(* Logix 5000 project; controller PBS_Perfusion vendor 1 type 14 code 217 rev 32.14; software revision 32.03; part 16 of 27 *)
(* tags used below, declared in another part *)
   Inp_IOFault : BOOL;   // Input Communication Status 0=OK, 1=fail
   Inp_Sim : BOOL;   // 1=Simulate working device; 0=Turn ON/OFF actual device
   Inp_OvrdCmd : DINT;   // Ovrd Device Command 0=None, 1=Off, 2=On, 3=Pulse Off, 4=Pulse On, 5=Pulse Cont
   Cfg_HasOnFdbk : BOOL;   // 1=Device provides an ON feedback signal
   Cfg_HasOffFdbk : BOOL;   // 1=Device provides an OFF feedback signal
   PSet_Owner : DINT;   // Program Owner Request ID (non-zero) or Release (zero)
   PCmd_On : BOOL;   // Program Command to turn device ON
   PCmd_Off : BOOL;   // Program Command to turn device OFF
   PCmd_OnPulse : BOOL;   // Program Command to pulse device (which is OFF) ON once
   PCmd_OffPulse : BOOL;   // Program Command to pulse device (which is ON) OFF once
   PCmd_ContPulse : BOOL;   // Program Command to pulse device continuously (blink)
   XCmd_On : BOOL;   // External Command to turn device ON
   XCmd_Off : BOOL;   // External Command to turn device OFF
   XCmd_OnPulse : BOOL;   // External Command to pulse device (which is OFF) ON once
   XCmd_OffPulse : BOOL;   // External Command to pulse device (which is ON) OFF once
   XCmd_ContPulse : BOOL;   // External Command to pulse device continuously (blink)
   XCmd_Reset : BOOL;   // Ext Cmd to clear shed latches and cleared alarms
   Out_Horn : BOOL;   // 1=Sound audible prior to commanded energize/ state change
   SrcQ_IO : DINT;   // Source and Quality of primary I/O (enumeration)
   SrcQ : DINT;   // Source and Quality of primary Val/Sts (enumeration)
   Val_Cmd : DINT;   // Device Command: 0=None, 1=Off, 2=On, 3=Pulse Off, 4=Pulse On, 5=Pulse Cont
   Val_Sts : DINT;   // Device Status 0=off 1=on 2=pulse off 3=pulse on 4=pulse cont. 5=turning off 6=turning on
   Val_Fault : DINT;   // Device Fault Status 0=none, 16=Feedback Fault, 32=I/O Fault, 34=Config Error
   Val_State : DINT;   // Internal Logic State (for animating STD on faceplate), see manual
   Val_NotifyAll : DINT;   // Highest Alarm prio and ack status this object + attached (enum)
   Val_UnackAlmC : DINT;   // Count of Unacknowledged Alarms
   Val_Owner : DINT;   // Current Object Owner ID (0=not owned)
   Sts_Out : BOOL;   // 1=Output is ON (energized), 0=Output is OFF (de-energized)
   Sts_Horn : BOOL;   // 1=Horn Active
   Nrdy_CfgErr : BOOL;   // 1=Device Not Ready: Configuration Error
   Nrdy_Fail : BOOL;   // 1=Device Not Ready: Device Failure (Shed Requires Reset)
   Nrdy_IOFault : BOOL;   // 1=Device Not Ready: I/O Fault (Shed Requires Reset)
   Nrdy_PrioOff : BOOL;   // 1=Device Not Ready: Oper/Ext Priority Off Comand Requires Reset
   Sts_AlmInh : BOOL;   // 1=One or more Alarms Shelved, Disabled or Suppressed
   Err_Alarm : BOOL;   // 1=Error in Config: Alarm Min On Time, Shelf Time, Severity
   Sts_OoS : ALIAS FOR CmdSrc.Sts_OoS;
   Sts_RdyAck : BOOL;   // 1=An alarm is ready to be acknowledged
   Sts_OnFail : ALIAS FOR OnFail.Inp;   // 1=Device Failed to Turn ON
   Sts_OffFail : ALIAS FOR OffFail.Inp;   // 1=Device Failed to Turn OFF
   Sts_IOFault : ALIAS FOR IOFault.Inp;   // I/O Comm Fault Status (0=OK, 1=Bad)
   P_DOut : BOOL;   // Unique Parameter Name for auto - discovery
   Wrk_Notify : DINT;   // Buffer for building Val_Notify
   CmdSrc : P_CmdSrc;   // Control / Command Source Selection
   IOFault : P_Alarm;   // I/O Fault Alarm
   IntlkTrip : P_Alarm;   // Interlock Trip Alarm
   OffFail : P_Alarm;   // Device Failed to Turn OFF Alarm
   OnFail : P_Alarm;   // Device Failed to Turn ON Alarm
   Wrk_Cmd : DINT;   // Device Command: 0= None, bit .0=Off, bit .1=On, bit .2=Pulse Off, bit .3=Pulse On, bit .4=Pulse Cont.
   Wrk_Fault : DINT;   // Buffer for building Val_Fault
   Wrk_SrcQ : DINT;   // Register for building Source / Quality enumeration
   Wrk_UnackAlmC : DINT;   // Buffer for building Val_UnackAlmC
   Val_Notify : DINT;   // Current Alarm Level and Acknowledgement (enumeration)
   OCmd_ResetAckAll : BOOL;   // Operator Command to Reset all Alarms and latched Shed conditions
   OCmd_ContPulse : BOOL;   // Operator Command to pulse device continuously (blink)
   OCmd_OffPulse : BOOL;   // Operator Command to pulse device (which is ON) OFF once
   OCmd_OnPulse : BOOL;   // Operator Command to pulse device (which is OFF) ON once
   OCmd_Off : BOOL;   // Operator Command to turn device OFF
   OCmd_On : BOOL;   // Operator Command to turn device ON
   MCmd_Check : BOOL;   // Maintenance Command to Check (not bypass) all Interlocks and Permissives
   MCmd_Bypass : BOOL;   // Maintenance Command to Bypass all Bypassable Interlocks and Permissives
   ORdy_ResetAckAll : BOOL;   // 1=Ready for OCmd_ResetAckAll (enables HMI button)
   ORdy_ContPulse : BOOL;   // 1=Ready for OCmd_ContPulse (enables HMI button)
   ORdy_OffPulse : BOOL;   // 1=Ready for OCmd_OffPulse (enables HMI button)
   ORdy_OnPulse : BOOL;   // 1=Ready for OCmd_OnPulse (enables HMI button)
   ORdy_Off : BOOL;   // 1=Ready for OCmd_Off (enables HMI button)
   ORdy_On : BOOL;   // 1=Ready for OCmd_On (enables HMI button)
   MRdy_Check : BOOL;   // 1=Ready for MCmd_Check (enables HMI button)
   MRdy_Bypass : BOOL;   // 1=Ready for MCmd_Bypass (enables HMI button)
   Wrk_State : DINT;   // Internal value of state machine current state
   Wrk_StartHorn : BOOL;   // 1=Sound audible prior to commanded energize/ state change
   ONS : DINT[3];
   REAL : DINT;
(* P_DOut, continued *)

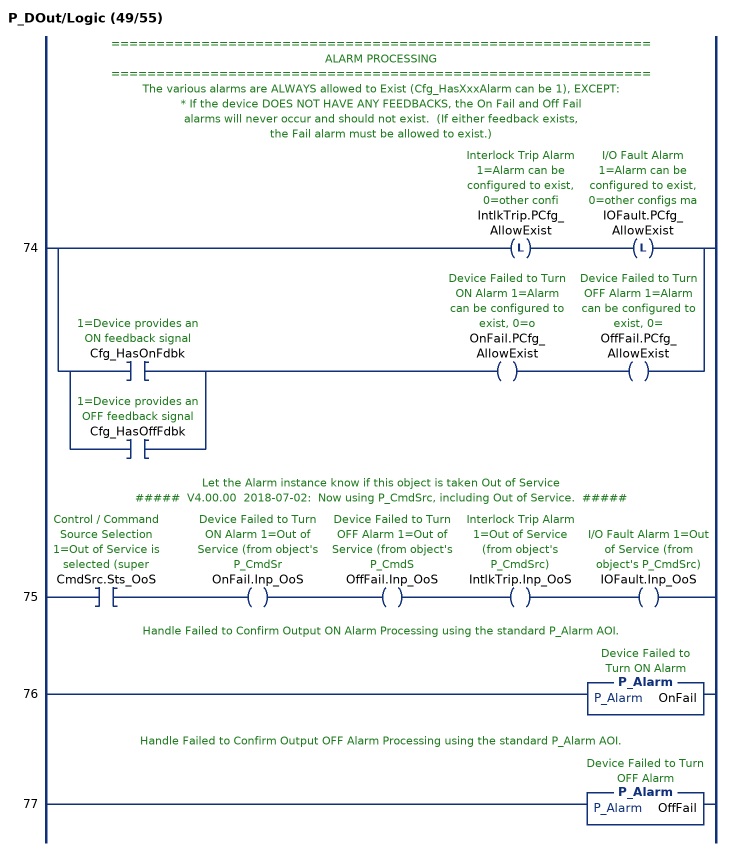
   // ============================================================
   // ALARM PROCESSING
   // ============================================================
   // The various alarms are ALWAYS allowed to Exist (Cfg_HasXxxAlarm can be 1), EXCEPT:
   // * If the device DOES NOT HAVE ANY FEEDBACKS, the On Fail and Off Fail
   // alarms will never occur and should not exist.  (If either feedback exists,
   // the Fail alarm must be allowed to exist.)
   74: [OTL(IntlkTrip.PCfg_AllowExist) OTL(IOFault.PCfg_AllowExist) ,[XIC(Cfg_HasOnFdbk) ,XIC(Cfg_HasOffFdbk) ] OTE(OnFail.PCfg_AllowExist) OTE(OffFail.PCfg_AllowExist) ];
   // Let the Alarm instance know if this object is taken Out of Service
   // #####  V4.00.00  2018-07-02:  Now using P_CmdSrc, including Out of Service.  #####
   75: XIC(CmdSrc.Sts_OoS)OTE(OnFail.Inp_OoS)OTE(OffFail.Inp_OoS)OTE(IntlkTrip.Inp_OoS)OTE(IOFault.Inp_OoS);
   // Handle Failed to Confirm Output ON Alarm Processing using the standard P_Alarm AOI.
   76: P_Alarm(OnFail);
   // Handle Failed to Confirm Output OFF Alarm Processing using the standard P_Alarm AOI.
   77: P_Alarm(OffFail);
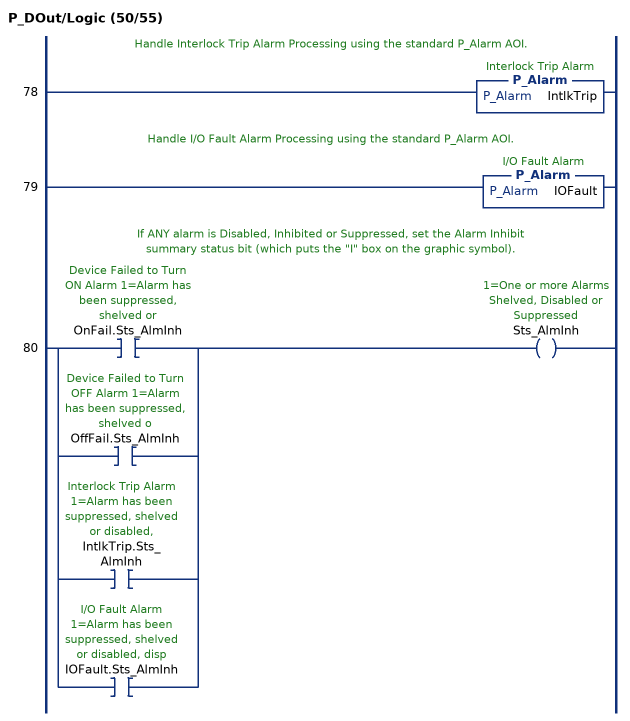
   // Handle Interlock Trip Alarm Processing using the standard P_Alarm AOI.
   78: P_Alarm(IntlkTrip);
   // Handle I/O Fault Alarm Processing using the standard P_Alarm AOI.
   79: P_Alarm(IOFault);
   // If ANY alarm is Disabled, Inhibited or Suppressed, set the Alarm Inhibit
   // summary status bit (which puts the "I" box on the graphic symbol).
   80: [XIC(OnFail.Sts_AlmInh) ,XIC(OffFail.Sts_AlmInh) ,XIC(IntlkTrip.Sts_AlmInh) ,XIC(IOFault.Sts_AlmInh) ]OTE(Sts_AlmInh);
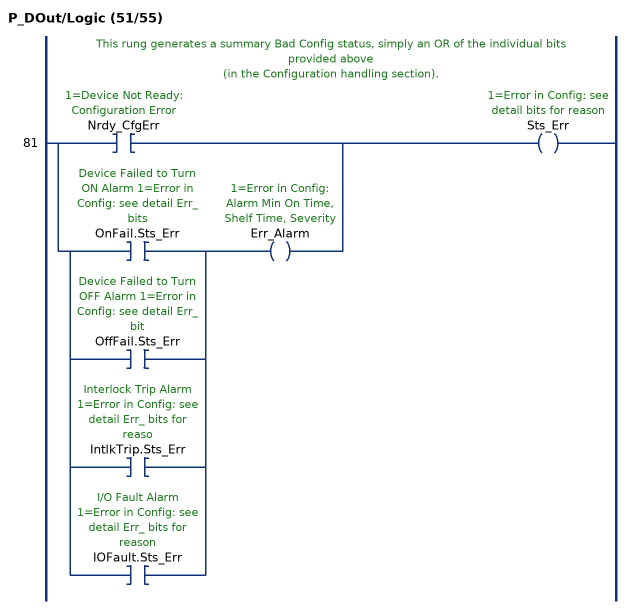
   // This rung generates a summary Bad Config status, simply an OR of the individual bits provided above
   // (in the Configuration handling section).
   81: [XIC(Nrdy_CfgErr) ,[XIC(OnFail.Sts_Err) ,XIC(OffFail.Sts_Err) ,XIC(IntlkTrip.Sts_Err) ,XIC(IOFault.Sts_Err) ] OTE(Err_Alarm) ]OTE(Sts_Err);
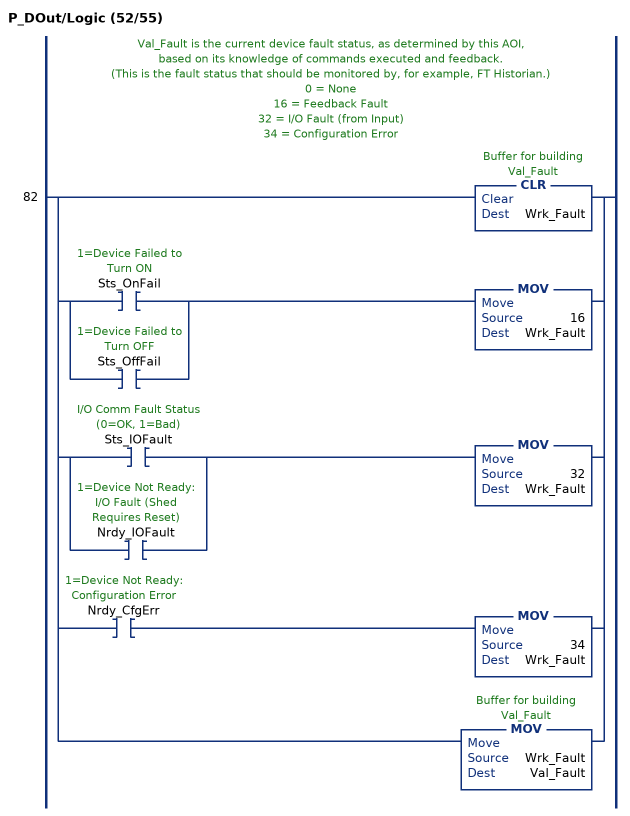
   // Val_Fault is the current device fault status, as determined by this AOI,
   // based on its knowledge of commands executed and feedback.
   // (This is the fault status that should be monitored by, for example, FT Historian.)
   // 0 = None
   // 16 = Feedback Fault
   // 32 = I/O Fault (from Input)
   // 34 = Configuration Error
   82: [CLR(Wrk_Fault) ,[XIC(Sts_OnFail) ,XIC(Sts_OffFail) ] MOV(16,Wrk_Fault) ,[XIC(Sts_IOFault) ,XIC(Nrdy_IOFault) ] MOV(32,Wrk_Fault) ,XIC(Nrdy_CfgErr) MOV(34,Wrk_Fault) ,MOV(Wrk_Fault,Val_Fault) ];
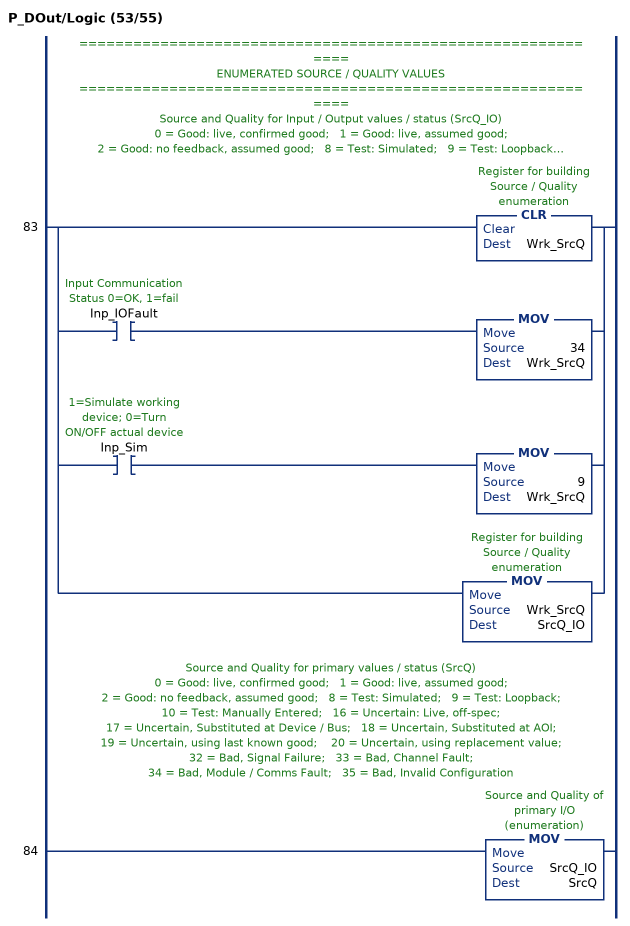
   // ============================================================
   // ENUMERATED SOURCE / QUALITY VALUES
   // ============================================================
   // Source and Quality for Input / Output values / status (SrcQ_IO)
   // 0 = Good: live, confirmed good;   1 = Good: live, assumed good;
   // 2 = Good: no feedback, assumed good;   8 = Test: Simulated;   9 = Test: Loopback;
   // 10 = Test: Manually Entered;   16 = Uncertain: Live, off-spec;
   // 17 = Uncertain, Substituted at Device / Bus;   18 = Uncertain, Substituted at AOI;
   // 19 = Uncertain, using last known good;    20 = Uncertain, using replacement value;
   // 32 = Bad, Signal Failure;   33 = Bad, Channel Fault;
   // 34 = Bad, Module / Comms Fault;   35 = Bad, Invalid Configuration
   83: [CLR(Wrk_SrcQ) ,XIC(Inp_IOFault) MOV(34,Wrk_SrcQ) ,XIC(Inp_Sim) MOV(9,Wrk_SrcQ) ,MOV(Wrk_SrcQ,SrcQ_IO) ];
   // Source and Quality for primary values / status (SrcQ)
   // 0 = Good: live, confirmed good;   1 = Good: live, assumed good;
   // 2 = Good: no feedback, assumed good;   8 = Test: Simulated;   9 = Test: Loopback;
   // 10 = Test: Manually Entered;   16 = Uncertain: Live, off-spec;
   // 17 = Uncertain, Substituted at Device / Bus;   18 = Uncertain, Substituted at AOI;
   // 19 = Uncertain, using last known good;    20 = Uncertain, using replacement value;
   // 32 = Bad, Signal Failure;   33 = Bad, Channel Fault;
   // 34 = Bad, Module / Comms Fault;   35 = Bad, Invalid Configuration
   84: MOV(SrcQ_IO,SrcQ);
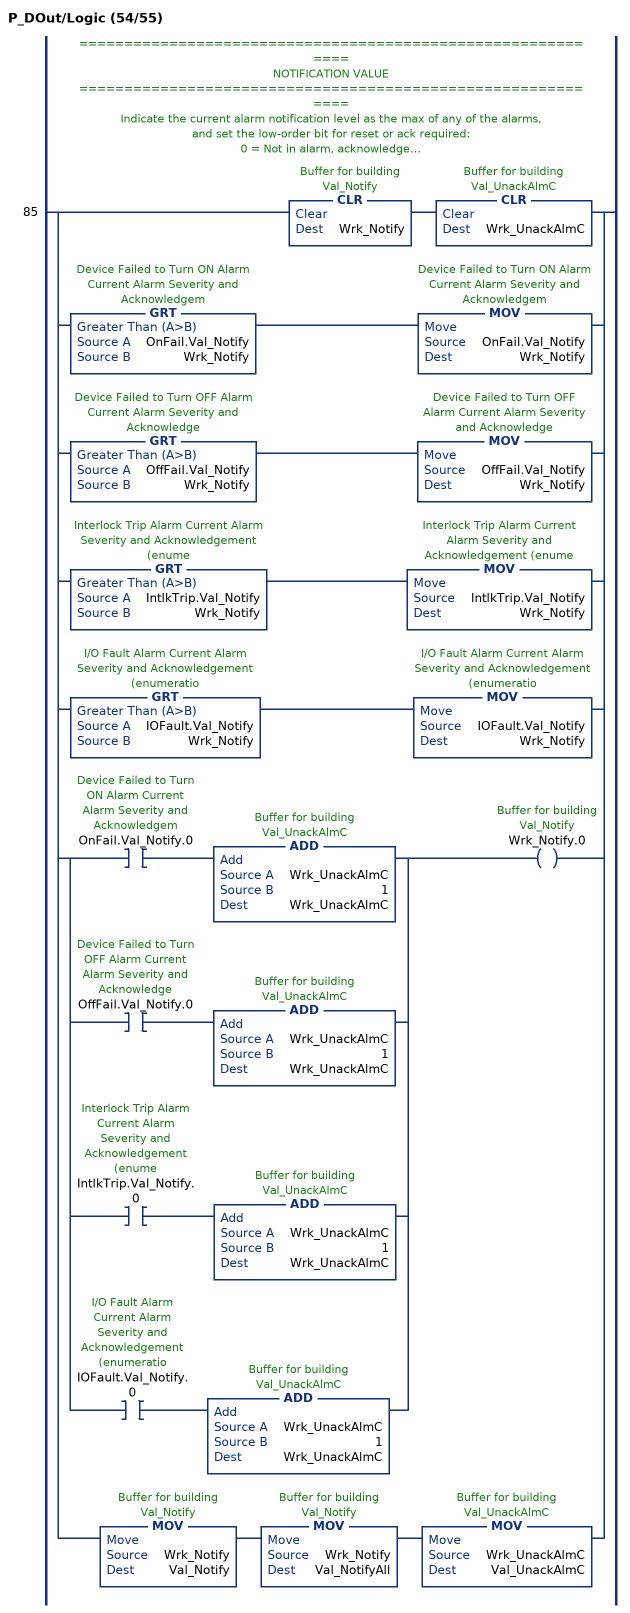
   // ============================================================
   // NOTIFICATION VALUE
   // ============================================================
   // Indicate the current alarm notification level as the max of any of the alarms,
   // and set the low-order bit for reset or ack required:
   // 0 = Not in alarm, acknowledged
   // 1 = Not in alarm, unacknowledged or reset required
   // 2 = Low severity alarm, acknowledged
   // 3 = Low severity alarm, unacknowledged
   // 4 = Medium severity alarm, acknowledged
   // 5 = Medium severity alarm, unacknowledged
   // 6 = High severity alarm, acknowledged
   // 7 = High severity alarm, unacknowledged
   // 8 = Urgent severity alarm, acknowledged
   // 9 = Urgent severity alarm, unacknowledged
   // #####  V4.00.00  2018-07-02:  Added Val_NotifyAll and Val_UnackAlmC to roll up alarm  #####
   // #####  priority / ack status and unack. alarm count.  #####
   85: [CLR(Wrk_Notify) CLR(Wrk_UnackAlmC) ,GRT(OnFail.Val_Notify,Wrk_Notify) MOV(OnFail.Val_Notify,Wrk_Notify) ,GRT(OffFail.Val_Notify,Wrk_Notify) MOV(OffFail.Val_Notify,Wrk_Notify) ,GRT(IntlkTrip.Val_Notify,Wrk_Notify) MOV(IntlkTrip.Val_Notify,Wrk_Notify) ,GRT(IOFault.Val_Notify,Wrk_Notify) MOV(IOFault.Val_Notify,Wrk_Notify) ,[XIC(OnFail.Val_Notify.0) ADD(Wrk_UnackAlmC,1,Wrk_UnackAlmC) ,XIC(OffFail.Val_Notify.0) ADD(Wrk_UnackAlmC,1,Wrk_UnackAlmC) ,XIC(IntlkTrip.Val_Notify.0) ADD(Wrk_UnackAlmC,1,Wrk_UnackAlmC) ,XIC(IOFault.Val_Notify.0) ADD(Wrk_UnackAlmC,1,Wrk_UnackAlmC) ] OTE(Wrk_Notify.0) ,MOV(Wrk_Notify,Val_Notify) MOV(Wrk_Notify,Val_NotifyAll) MOV(Wrk_UnackAlmC,Val_UnackAlmC) ];
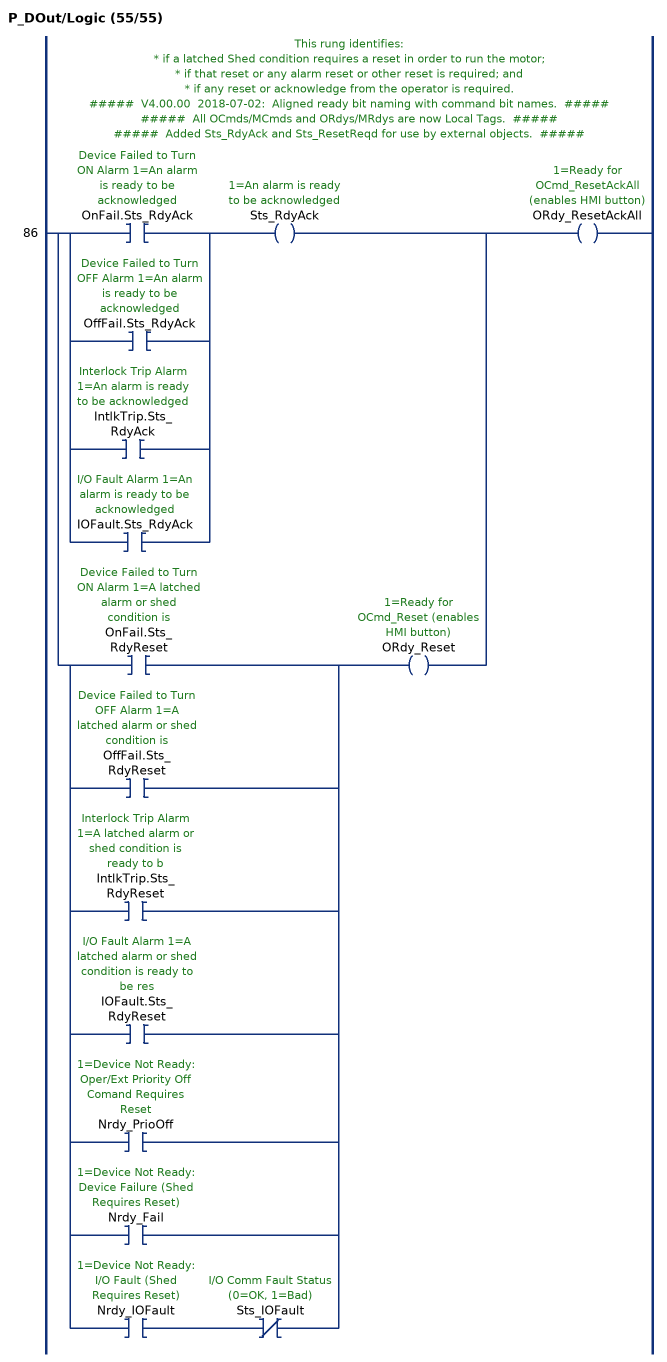
   // This rung identifies:
   // * if a latched Shed condition requires a reset in order to run the motor;
   // * if that reset or any alarm reset or other reset is required; and
   // * if any reset or acknowledge from the operator is required.
   // #####  V4.00.00  2018-07-02:  Aligned ready bit naming with command bit names.  #####
   // #####  All OCmds/MCmds and ORdys/MRdys are now Local Tags.  #####
   // #####  Added Sts_RdyAck and Sts_ResetReqd for use by external objects.  #####
   86: [[XIC(OnFail.Sts_RdyAck) ,XIC(OffFail.Sts_RdyAck) ,XIC(IntlkTrip.Sts_RdyAck) ,XIC(IOFault.Sts_RdyAck) ] OTE(Sts_RdyAck) ,[XIC(OnFail.Sts_RdyReset) ,XIC(OffFail.Sts_RdyReset) ,XIC(IntlkTrip.Sts_RdyReset) ,XIC(IOFault.Sts_RdyReset) ,XIC(Nrdy_PrioOff) ,XIC(Nrdy_Fail) ,XIC(Nrdy_IOFault) XIO(Sts_IOFault) ] OTE(ORdy_Reset) ]OTE(ORdy_ResetAckAll);
END_ROUTINE

ROUTINE Prescan   (* ladder *)
// Clear Ownershp, clear "lurking" Commands, de-energize output
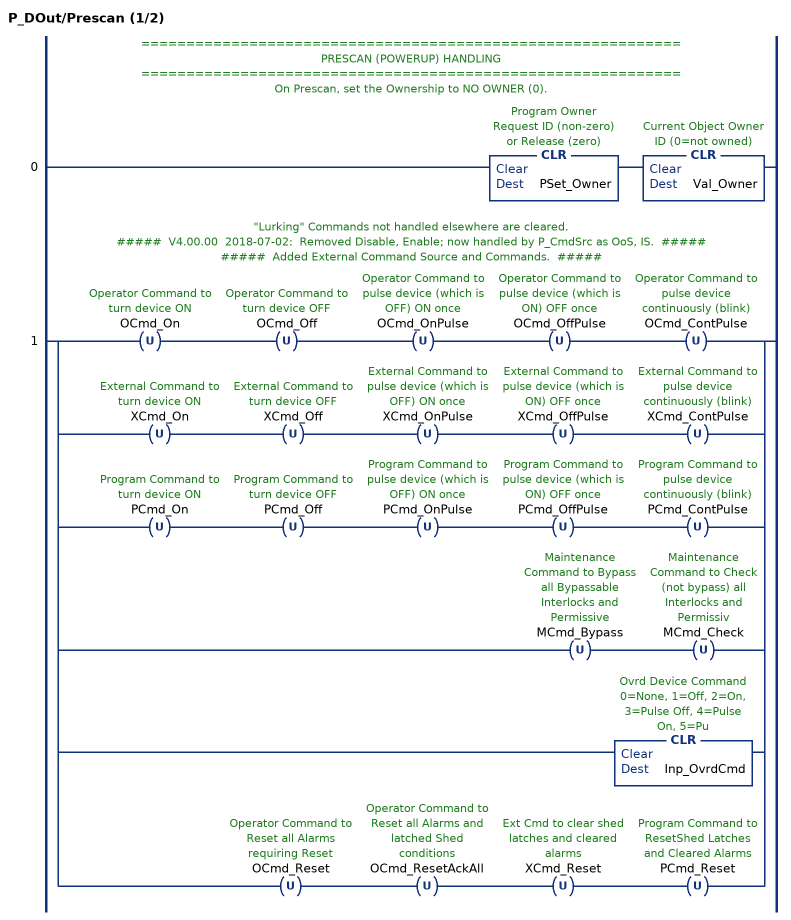
   // ============================================================
   // PRESCAN (POWERUP) HANDLING
   // ============================================================
   // On Prescan, set the Ownership to NO OWNER (0).
   0: CLR(PSet_Owner)CLR(Val_Owner);
   // "Lurking" Commands not handled elsewhere are cleared.
   // #####  V4.00.00  2018-07-02:  Removed Disable, Enable; now handled by P_CmdSrc as OoS, IS.  #####
   // #####  Added External Command Source and Commands.  #####
   1: [OTU(OCmd_On) OTU(OCmd_Off) OTU(OCmd_OnPulse) OTU(OCmd_OffPulse) OTU(OCmd_ContPulse) ,OTU(XCmd_On) OTU(XCmd_Off) OTU(XCmd_OnPulse) OTU(XCmd_OffPulse) OTU(XCmd_ContPulse) ,OTU(PCmd_On) OTU(PCmd_Off) OTU(PCmd_OnPulse) OTU(PCmd_OffPulse) OTU(PCmd_ContPulse) ,OTU(MCmd_Bypass) OTU(MCmd_Check) ,CLR(Inp_OvrdCmd) ,OTU(OCmd_Reset) OTU(OCmd_ResetAckAll) OTU(XCmd_Reset) OTU(PCmd_Reset) ];
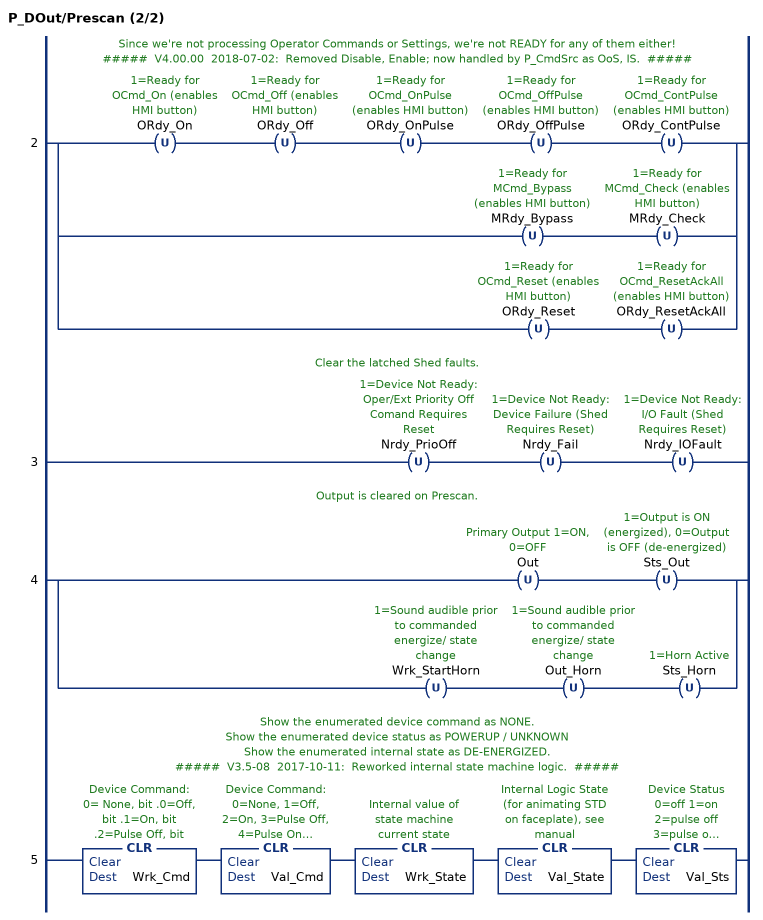
   // Since we're not processing Operator Commands or Settings, we're not READY for any of them either!
   // #####  V4.00.00  2018-07-02:  Removed Disable, Enable; now handled by P_CmdSrc as OoS, IS.  #####
   2: [OTU(ORdy_On) OTU(ORdy_Off) OTU(ORdy_OnPulse) OTU(ORdy_OffPulse) OTU(ORdy_ContPulse) ,OTU(MRdy_Bypass) OTU(MRdy_Check) ,OTU(ORdy_Reset) OTU(ORdy_ResetAckAll) ];
   // Clear the latched Shed faults.
   3: OTU(Nrdy_PrioOff)OTU(Nrdy_Fail)OTU(Nrdy_IOFault);
   // Output is cleared on Prescan.
   4: [OTU(Out) OTU(Sts_Out) ,OTU(Wrk_StartHorn) OTU(Out_Horn) OTU(Sts_Horn) ];
   // Show the enumerated device command as NONE.
   // Show the enumerated device status as POWERUP / UNKNOWN
   // Show the enumerated internal state as DE-ENERGIZED.
   // #####  V3.5-08  2017-10-11:  Reworked internal state machine logic.  #####
   5: CLR(Wrk_Cmd)CLR(Val_Cmd)CLR(Wrk_State)CLR(Val_State)CLR(Val_Sts);
END_ROUTINE
END_ADD_ON_INSTRUCTION

ADD_ON_INSTRUCTION P_Gate   (* revision 4.10 .00 Release, vendor Rockwell Automation, ExecutePrescan, ExecuteEnableInFalse *)
// Condition Gate/Delay
// Revision note:
// See Instruction Help for a summary of changes, and see 4.10 Release Notes for details.
// Help:
// Copyright © Rockwell Automation, Inc.  All Rights Reserved.
// This Instruction provides a "gate" for a discrete Input signal and
// provides on-delay and off-delay timing for the gated signal.
// When the Gate input is true, the instruction Input is passed through
// to the Output, with on-delay and off-delay timing applied.
// When the Gate input is false, the Output is kept off
// (note: off-delay still applies!)
// This instruction is usually used between a comparison
// (analog threshold with deadband or discrete logic)
// and a P_Alarm instance, but may be used as a
// gated on-delay/off-delay timer generally.
// When EnableIn  is FALSE (e.g., on a false LD rung), the Input "Inp"
// is inverted.  Note that the Gate input (Inp_Gate) is NOT inverted!!!
// SUMMARY OF CHANGES FROM PREVIOUS VERSION (4.00.00)
// See 4.10 Release Notes for details.
// * Unmodified, up-rev only for Library 4.10.00
// SUMMARY OF CHANGES FROM PREVIOUS VERSION (3.5-01)
// See 4.00 Release Notes for details.
// * Changed Inf_ items to HMI_ (e.g., HMI_Lib, HMI_Type).
// * Changed delay time configuration items to REAL seconds
VAR_INPUT
   Inp : BOOL; {visible}   // Input Condition: e.g., result of comparison
   Inp_Gate : BOOL := 1; {visible}   // Gate Input: 1=enable On Delay / Off Delay after Gate Delay, 0=disable
   Cfg_GateDly : REAL;   // Gate Delay (s): time after Gate Input true to enable On/Off Delay
   Cfg_OnDly : REAL;   // On Delay (s): If Gate Delay done, time Inp must be true to set Out true
   Cfg_OffDly : REAL;   // Off Delay (s): Time after Inp or Gate goes to 0 for Out to go to 0
END_VAR
VAR_OUTPUT
   Out : BOOL; {access Read Only, visible}   // Output after On Delay, Off Delay, enabled by Gate
   Sts_Gate : BOOL; {access Read Only, visible}   // 1=Gate Delay done, Output is enabled
   Sts_Err : BOOL; {access Read Only, visible}   // 1=Error in Config (see detail Err_ bits for reason), display icon
   Err_Timer : BOOL; {access Read Only}   // 1=Error in Config: On Delay, Off Delay, Gate Delay Time Invalid (use 0 to 2147483 s)
   P_Gate : BOOL;   // Unique Parameter Name for auto - discovery
END_VAR
VAR
   Wrk_OffDlyT : TIMER; {access Read Only}   // Off Delay Timer
   Wrk_OnDlyT : TIMER; {access Read Only}   // On Delay Timer
   Wrk_GateT : TIMER; {access Read Only}   // Gate Delay Timer
   Cfg_InpCond : STRING_20 := 'Input Condition';   // Displayed text of P_Gate's Input (Inp) Condition
   HMI_Lib : STRING_12 := 'RA-BAS'; {access Read Only}   // Display Library for Faceplate call-up
   HMI_Type : STRING_16 := 'P_Gate'; {access Read Only}   // Must contain AOI name, used for HMI and Information S/W
   Cfg_GateCond : STRING_20 := 'Gating Condition';   // Displayed text of P_Gate's Gating (Inp_Gate) Condition
   HMI_Tab : SINT;   // Tab to display (FTView ME)
END_VAR

ROUTINE EnableInFalse   (* ladder *)
// Same as main Logic routine, except Inp is inverted (for use in LD logic)  (Inp_Gate is NOT inverted!!!)
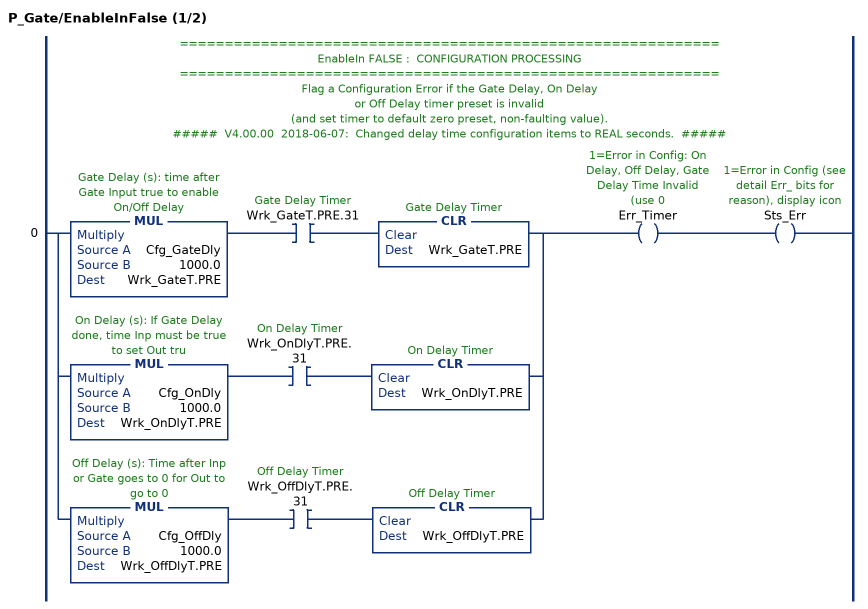
   // ============================================================
   // EnableIn FALSE :  CONFIGURATION PROCESSING
   // ============================================================
   // Flag a Configuration Error if the Gate Delay, On Delay
   // or Off Delay timer preset is invalid
   // (and set timer to default zero preset, non-faulting value).
   // #####  V4.00.00  2018-06-07:  Changed delay time configuration items to REAL seconds.  #####
   0: [MUL(Cfg_GateDly,1000.0,Wrk_GateT.PRE) XIC(Wrk_GateT.PRE.31) CLR(Wrk_GateT.PRE) ,MUL(Cfg_OnDly,1000.0,Wrk_OnDlyT.PRE) XIC(Wrk_OnDlyT.PRE.31) CLR(Wrk_OnDlyT.PRE) ,MUL(Cfg_OffDly,1000.0,Wrk_OffDlyT.PRE) XIC(Wrk_OffDlyT.PRE.31) CLR(Wrk_OffDlyT.PRE) ]OTE(Err_Timer)OTE(Sts_Err);
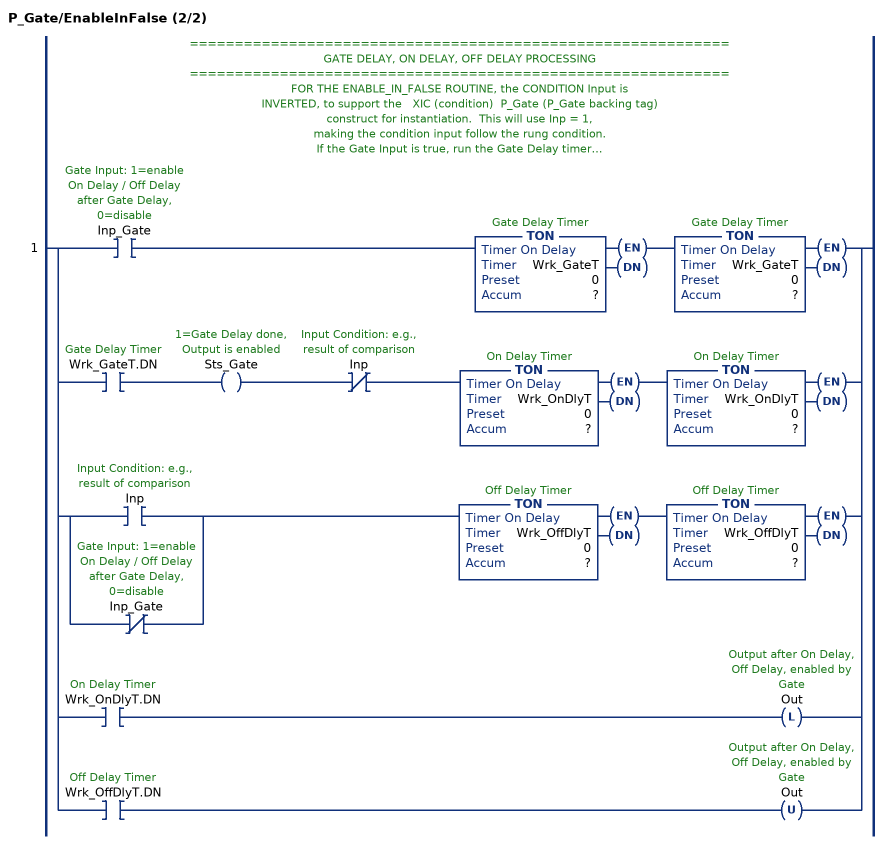
   // ============================================================
   // GATE DELAY, ON DELAY, OFF DELAY PROCESSING
   // ============================================================
   // FOR THE ENABLE_IN_FALSE ROUTINE, the CONDITION Input is
   // INVERTED, to support the   XIC (condition)  P_Gate (P_Gate backing tag)
   // construct for instantiation.  This will use Inp = 1,
   // making the condition input follow the rung condition.
   // If the Gate Input is true, run the Gate Delay timer.
   // Once the Gate Delay is complete, enable the
   // On Delay and Off Delay that follow the INVERTED input.
   // Report the Gate Delay status and the final Output status (after all delays).
   // @@@@@  NOTE: Doubled TONs are used to ensure that  @@@@@
   // @@@@@  .DN bit transitions on same scan if Preset = 0 !  @@@@@
   1: [XIC(Inp_Gate) TON(Wrk_GateT,?,?) TON(Wrk_GateT,?,?) ,XIC(Wrk_GateT.DN) OTE(Sts_Gate) XIO(Inp) TON(Wrk_OnDlyT,?,?) TON(Wrk_OnDlyT,?,?) ,[XIC(Inp) ,XIO(Inp_Gate) ] TON(Wrk_OffDlyT,?,?) TON(Wrk_OffDlyT,?,?) ,XIC(Wrk_OnDlyT.DN) OTL(Out) ,XIC(Wrk_OffDlyT.DN) OTU(Out) ];
END_ROUTINE

ROUTINE Logic   (* ladder *)
// Gate the input and apply on-delay and off-delay timing
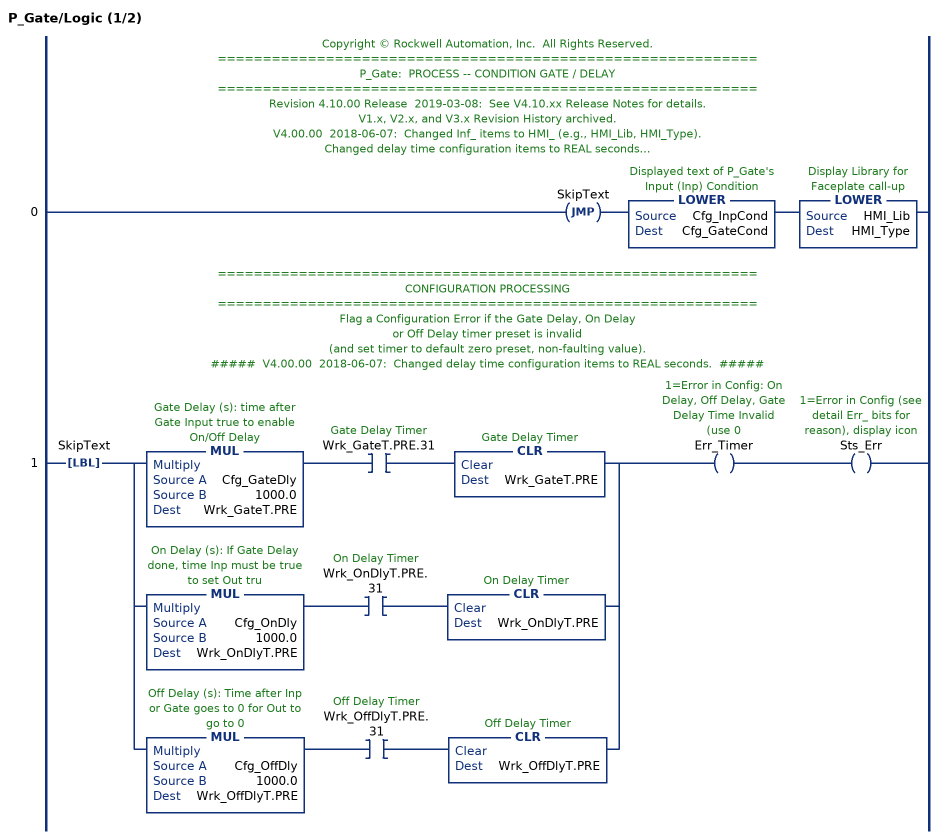
   // Copyright © Rockwell Automation, Inc.  All Rights Reserved.
   // ============================================================
   // P_Gate:  PROCESS -- CONDITION GATE / DELAY
   // ============================================================
   // Revision 4.10.00 Release  2019-03-08:  See V4.10.xx Release Notes for details.
   // V1.x, V2.x, and V3.x Revision History archived.
   // V4.00.00  2018-06-07:  Changed Inf_ items to HMI_ (e.g., HMI_Lib, HMI_Type).
   // Changed delay time configuration items to REAL seconds.
   // V4.10.00  2019-03-08:  Unmodified, up-rev only for Library 4.10.00
   // ============================================================
   // This Instruction provides a "gate" for a discrete Input signal and
   // provides on-delay and off-delay timing for the gated signal.
   // When the Gate input is true, the instruction Input is passed through
   // to the Output, with on-delay and off-delay timing applied.
   // When the Gate input is false, the Output is kept off
   // (note: off-delay still applies!)
   // This instruction is usually used between a comparison
   // (analog threshold with deadband or discrete logic)
   // and a P_Alarm instance, but may be used as a
   // gated on-delay/off-delay timer generally.
   // When EnableIn  is FALSE (e.g., on a false LD rung),
   // the Input "Inp" is inverted.  Note that the Gate
   // input (Inp_Gate) is NOT inverted!!!
   // ============================================================
   // SHOW LOCAL STRINGS
   // ============================================================
   // The STRINGs containing the text associated with each instance of this
   // instruction cannot be Input or Output Parameters, because STRINGs are not
   //  'atomic' types. (Inputs and Outputs must be SINT, INT, DINT, REAL, or BOOL.)
   // In order to make it easier to find and configure these STRINGs, this rung
   // was added.  THE JMP (and the LBL on the following rung)
   // MUST NOT BE REMOVED!!!
   // To view the STRINGs, go to the instruction instance (in LD or FBD), RIGHT-click
   // to bring up the context menu and select "Open Instruction Logic".
   // This rung will appear with the STRING values for the selected instance.
   // You may double-click the STRING values here to modify them as well.
   0: JMP(SkipText)LOWER(Cfg_InpCond,Cfg_GateCond)LOWER(HMI_Lib,HMI_Type);
   // ============================================================
   // CONFIGURATION PROCESSING
   // ============================================================
   // Flag a Configuration Error if the Gate Delay, On Delay
   // or Off Delay timer preset is invalid
   // (and set timer to default zero preset, non-faulting value).
   // #####  V4.00.00  2018-06-07:  Changed delay time configuration items to REAL seconds.  #####
   1: LBL(SkipText)[MUL(Cfg_GateDly,1000.0,Wrk_GateT.PRE) XIC(Wrk_GateT.PRE.31) CLR(Wrk_GateT.PRE) ,MUL(Cfg_OnDly,1000.0,Wrk_OnDlyT.PRE) XIC(Wrk_OnDlyT.PRE.31) CLR(Wrk_OnDlyT.PRE) ,MUL(Cfg_OffDly,1000.0,Wrk_OffDlyT.PRE) XIC(Wrk_OffDlyT.PRE.31) CLR(Wrk_OffDlyT.PRE) ]OTE(Err_Timer)OTE(Sts_Err);
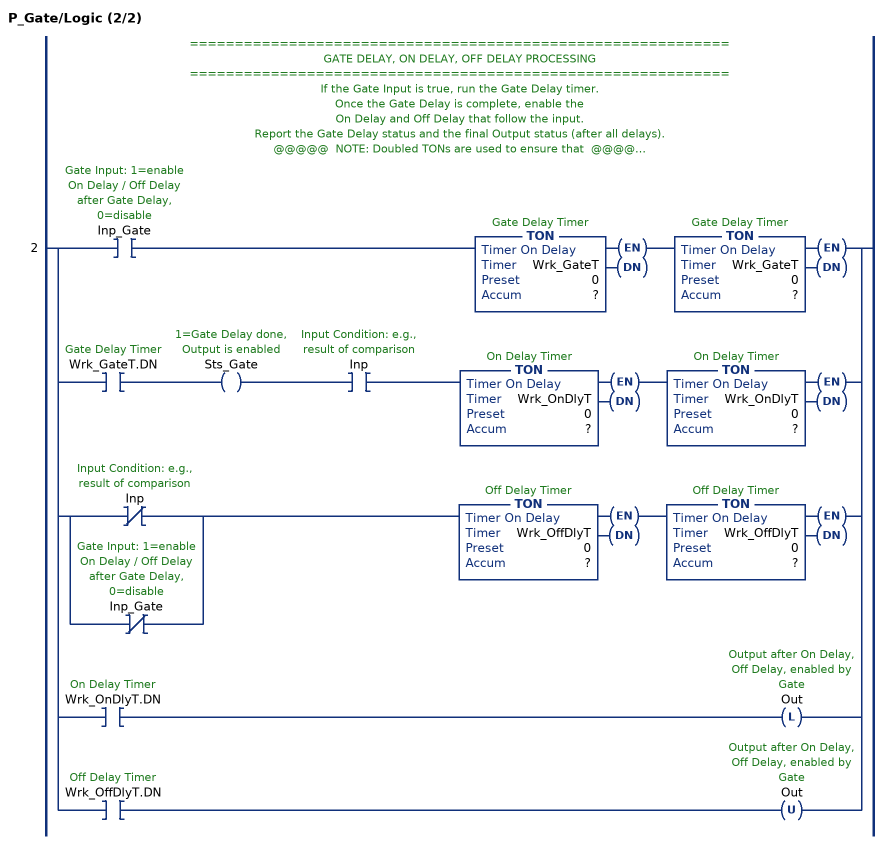
   // ============================================================
   // GATE DELAY, ON DELAY, OFF DELAY PROCESSING
   // ============================================================
   // If the Gate Input is true, run the Gate Delay timer.
   // Once the Gate Delay is complete, enable the
   // On Delay and Off Delay that follow the input.
   // Report the Gate Delay status and the final Output status (after all delays).
   // @@@@@  NOTE: Doubled TONs are used to ensure that  @@@@@
   // @@@@@  .DN bit transitions on same scan if Preset = 0 !  @@@@@
   2: [XIC(Inp_Gate) TON(Wrk_GateT,?,?) TON(Wrk_GateT,?,?) ,XIC(Wrk_GateT.DN) OTE(Sts_Gate) XIC(Inp) TON(Wrk_OnDlyT,?,?) TON(Wrk_OnDlyT,?,?) ,[XIO(Inp) ,XIO(Inp_Gate) ] TON(Wrk_OffDlyT,?,?) TON(Wrk_OffDlyT,?,?) ,XIC(Wrk_OnDlyT.DN) OTL(Out) ,XIC(Wrk_OffDlyT.DN) OTU(Out) ];
END_ROUTINE

ROUTINE Prescan   (* ladder *)
// Set the Gate Input to 1 (default value) on prescan
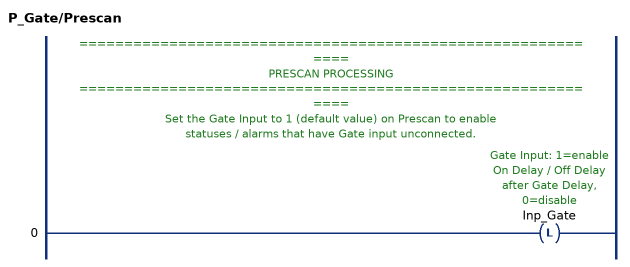
   // ============================================================
   // PRESCAN PROCESSING
   // ============================================================
   // Set the Gate Input to 1 (default value) on Prescan to enable
   // statuses / alarms that have Gate input unconnected.
   0: OTL(Inp_Gate);
END_ROUTINE
END_ADD_ON_INSTRUCTION

ADD_ON_INSTRUCTION P_Intlk   (* revision 4.10 .01 Release, vendor Rockwell Automation, ExecutePrescan, ExecuteEnableInFalse *)
// Interlocks
// Revision note:
// See Instruction Help for a summary of changes, and see 4.10 Release Notes for details.
// Help:
// Copyright © Rockwell Automation, Inc.  All Rights Reserved.
// This Instruction monitors up to 16 Interlock conditions.  It provides these features:
// *  The "OK" state of each Interlock Input is configurable.  By default,
//     each Input is 1 to trip, 0 when OK to run.
// *  Interlocks may be configured as Latched.  Latched Interlocks
//     require a Reset Command to clear.  The latching function can be
//     inhibited via a Latch Defeat input, for example, to avoid latching
//     Interlocks for a stopped motor.
// *  Interlocks may be configured as Bypassable; Non-Bypassable
//     Interlocks are reported separately so the destination object can
//     decide whether to bypass (ignore) bypassable interlocks, such
//     as in Maintenance Mode.
// *  First-Out reporting indicates the first condition that caused the
//     running equipment to be tripped.
// *  For each Interlock condition, a Tag may be defined for navigation.
//     Clicking the Interlock description will call up the associated Tag's
//     Faceplate.
// SUMMARY OF CHANGES FROM PREVIOUS VERSION (4.10.00)
// See 4.10 Release Notes for details.
// * Modified conditions for clearing first-out status and text.
// SUMMARY OF CHANGES FROM PREVIOUS VERSION (4.00.00)
// See 4.10 Release Notes for details.
// * Changed type of Val_FirstOutTxt to STRING_Cond.
// * Corrected Scan Mode selection to execute Prescan logic.
// * Added Cfg_HasMoreObj.
// SUMMARY OF CHANGES FROM PREVIOUS VERSION (3.5-05)
// See 4.00 Release Notes for details.
// * Changed Inf_ items to HMI_, and added Cfg_Area for security.
// * Added Val_FirstOutTxt string (Local, read-only) for use in
//    IntlkTrip alarm message  (ref: KnowledgeBase answer ID 672568).
// * Deleted Cfg_PCmdClear; all Program Commands are now self-clearing.
// * All OCmds/MCmds and ORdys/MRdys are now Local Tags.
// * Added Sts_RdyReset for use by external objects.
VAR_INPUT
   Inp_Intlk00 : ALIAS FOR Wrk_Inp.0; {visible}   // Interlock Cond. 00, Stop if not in configured OK state
   Inp_Intlk01 : ALIAS FOR Wrk_Inp.1; {visible}   // Interlock Cond. 01, Stop if not in configured OK state
   Inp_Intlk02 : ALIAS FOR Wrk_Inp.2; {visible}   // Interlock Cond. 02, Stop if not in configured OK state
   Inp_Intlk03 : ALIAS FOR Wrk_Inp.3; {visible}   // Interlock Cond. 03, Stop if not in configured OK state
   Inp_Intlk04 : ALIAS FOR Wrk_Inp.4; {visible}   // Interlock Cond. 04, Stop if not in configured OK state
   Inp_Intlk05 : ALIAS FOR Wrk_Inp.5; {visible}   // Interlock Cond. 05, Stop if not in configured OK state
   Inp_Intlk06 : ALIAS FOR Wrk_Inp.6; {visible}   // Interlock Cond. 06, Stop if not in configured OK state
   Inp_Intlk07 : ALIAS FOR Wrk_Inp.7; {visible}   // Interlock Cond. 07, Stop if not in configured OK state
   Inp_Intlk08 : ALIAS FOR Wrk_Inp.8;   // Interlock Cond. 08, Stop if not in configured OK state
   Inp_Intlk09 : ALIAS FOR Wrk_Inp.9;   // Interlock Cond. 09, Stop if not in configured OK state
   Inp_Intlk10 : ALIAS FOR Wrk_Inp.10;   // Interlock Cond. 10, Stop if not in configured OK state
   Inp_Intlk11 : ALIAS FOR Wrk_Inp.11;   // Interlock Cond. 11, Stop if not in configured OK state
   Inp_Intlk12 : ALIAS FOR Wrk_Inp.12;   // Interlock Cond. 12, Stop if not in configured OK state
   Inp_Intlk13 : ALIAS FOR Wrk_Inp.13;   // Interlock Cond. 13, Stop if not in configured OK state
   Inp_Intlk14 : ALIAS FOR Wrk_Inp.14;   // Interlock Cond. 14, Stop if not in configured OK state
   Inp_Intlk15 : ALIAS FOR Wrk_Inp.15;   // Interlock Cond. 15, Stop if not in configured OK state
   Inp_BypActive : BOOL; {visible}   // 1=Interlock Bypassing is currently active
   Inp_LatchDefeat : BOOL; {visible}   // Latch Defeat 1=Do not latch inputs even if configured for latching
   Inp_Reset : BOOL; {visible}   // 1=Reset Latched Interlocks and First-Out
   Cfg_OKState : INT;   // Bits indicate which state (0 or 1) of each input is OK to run
   Cfg_Latched : INT;   // Set bits indicate which conditions are latched (sealed in)
   Cfg_Bypassable : INT;   // Set bits indicate which conditions can be bypassed
   Cfg_HasNav : INT;   // Set bits indicate which Navigation buttons are enabled
   Cfg_HasMoreObj : BOOL;   // 1=Tells HMI an object with more info is available
   PCmd_Reset : BOOL;   // Program Command to Reset Latched Interlocks
END_VAR
VAR_OUTPUT
   Sts_IntlkOK : BOOL := 1; {access Read Only, visible}   // Overall Interlock Status (1=OK to run, 0=Stop)
   Sts_NBIntlkOK : BOOL := 1; {access Read Only, visible}   // Non-Bypassable Interlock Status (1=All NB Interlocks OK to run)
   Sts_BypActive : BOOL; {access Read Only}   // 1=Interlock Bypassing is Active (ignore bypassable interlocks)
   Sts_RdyReset : ALIAS FOR ORdy_Reset; {access Read Only}   // 1=A latched interlock (returned to OK) is ready to be reset
   Sts_Intlk : INT; {access Read Only, visible}   // Individual Interlock Status (1=Stop, 0=OK)
   Sts_FirstOut : INT; {access Read Only, visible}   // Interlock First Out Status (bit 1 is First Not-OK condition)
   P_Intlk : BOOL;   // Unique Parameter Name for auto - discovery
END_VAR
VAR
   Cfg_CondTxt : STRING_Cond[16] := ([0] := 'Enter Description #0');   // Short HMI description of Interlock Conditions
   Wrk_Inp : INT;   // Collection copy of Inp_IntlkXXs
   Wrk_NB : INT; {access None}   // Working register for Non-Bypassable Interlock ogic
   Wrk_Intlk : INT; {access None}   // Working register for Interlock logic
   Wrk_FirstOut : INT; {access None}   // Working register for First Out logic
   Wrk_Sts : INT; {access None}   // Working register for generating Interlock status
   Wrk_PrevSts : INT; {access None}   // Interlock Status previous scan
   Wrk_LatchEnable : BOOL := 1; {access None}   // 1=Latch interlock if configured to latch, 0=don't latch
   HMI_Tab : SINT;   // Tab to display (FTView ME)
   Wrk_InpInv : INT; {access None}   // Input states after inversion based on Cfg_OKState
   HMI_Type : STRING_16 := 'P_Intlk'; {access Read Only}   // Type identifier for HMI navigation
   Cfg_Label : STRING_20 := 'Interlocks';   // Label for graphic symbol displayed on HMI
   Cfg_Tag : STRING_20 := 'P_Intlk';   // Tagname for display on HMI
   Cfg_Desc : STRING_40 := 'Interlocks with First Out';   // Description for display on HMI
   Cfg_NavTag : STRING_NavTag[16];   // Tagnames for destinations of Navigation buttons
   HMI_Lib : STRING_12 := 'RA-BAS'; {access Read Only}   // Display Library for Faceplate call-up
   MSet_Bypass : INT;   // Individual condition Maintenance Bypass toggles
   Cfg_Area : STRING_Area := 'area01';   // Process Area for security
   Val_FirstOutTxt : STRING_Cond; {access Read Only}   // Text Description of First-Out Condition
   Wrk_NonIntlkStop : BOOL; {access None}   // One-Shot store: Stop OTHER than Interlock Stop occurred.
   Wrk_SetFirstOut : BOOL; {access None}   // One-Shot store: First Out update triggered
   ORdy_Reset : BOOL; {access Read Only}   // 1=Ready for OCmd_Reset (enables HMI button)
   OCmd_Reset : BOOL;   // Operator Command to Reset Latched Interlocks
END_VAR

ROUTINE EnableInFalse   (* ladder *)
// Set summary "OK" Status bits to FALSE (0)
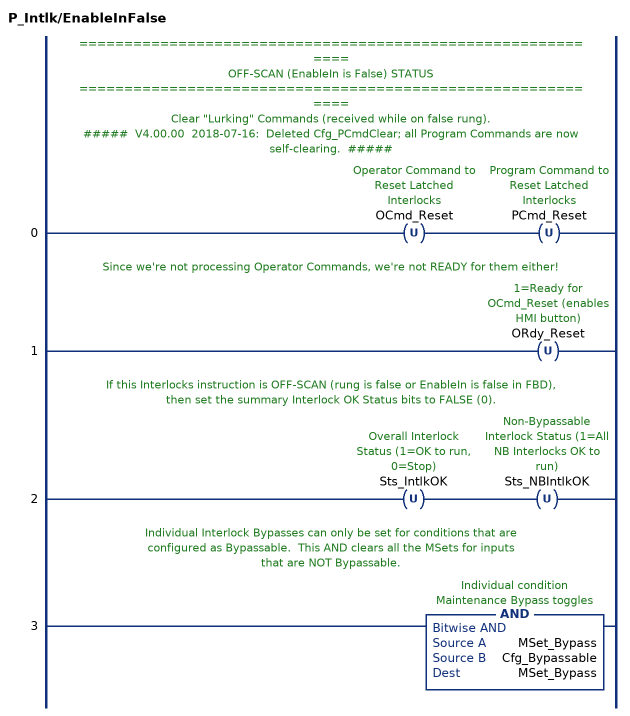
   // ============================================================
   // OFF-SCAN (EnableIn is False) STATUS
   // ============================================================
   //  Clear "Lurking" Commands (received while on false rung).
   // #####  V4.00.00  2018-07-16:  Deleted Cfg_PCmdClear; all Program Commands are now self-clearing.  #####
   0: OTU(OCmd_Reset)OTU(PCmd_Reset);
   // Since we're not processing Operator Commands, we're not READY for them either!
   1: OTU(ORdy_Reset);
   // If this Interlocks instruction is OFF-SCAN (rung is false or EnableIn is false in FBD),
   // then set the summary Interlock OK Status bits to FALSE (0).
   2: OTU(Sts_IntlkOK)OTU(Sts_NBIntlkOK);
   // Individual Interlock Bypasses can only be set for conditions that are
   // configured as Bypassable.  This AND clears all the MSets for inputs
   // that are NOT Bypassable.
   3: AND(MSet_Bypass,Cfg_Bypassable,MSet_Bypass);
END_ROUTINE

ROUTINE Logic   (* ladder *)
// Check Interlock Conditions
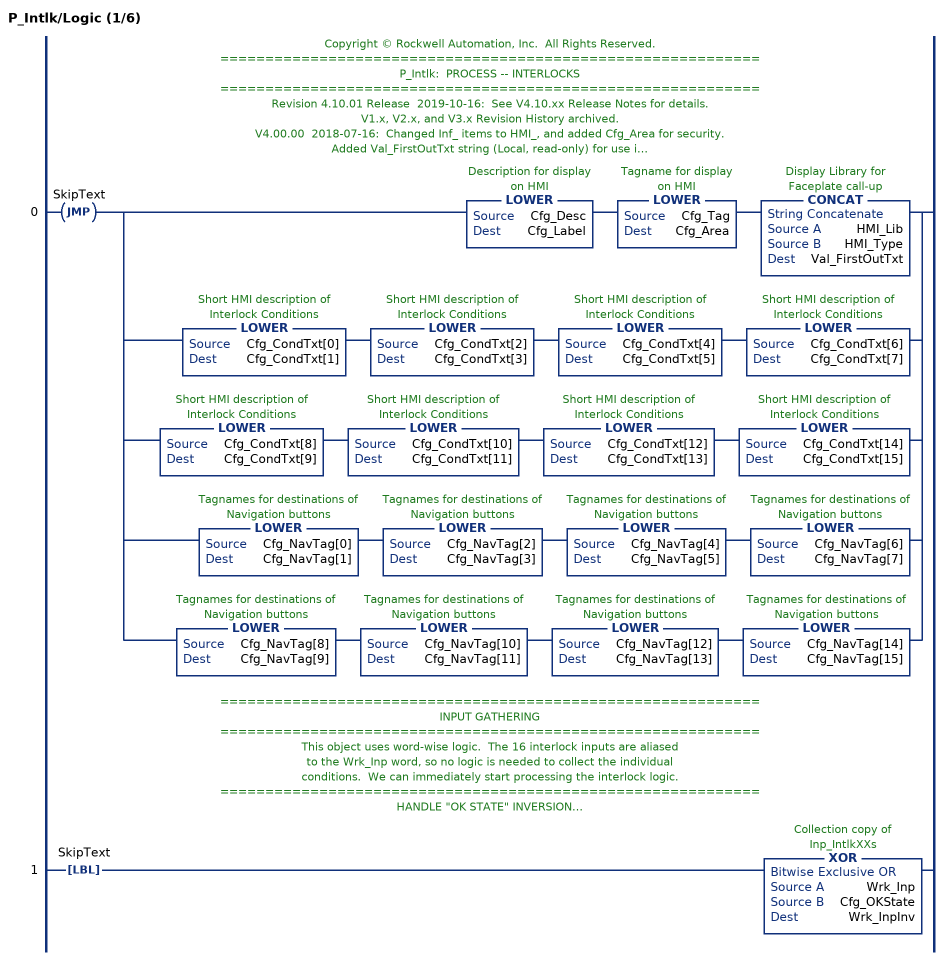
   // Copyright © Rockwell Automation, Inc.  All Rights Reserved.
   // ============================================================
   // P_Intlk:  PROCESS -- INTERLOCKS
   // ============================================================
   // Revision 4.10.01 Release  2019-10-16:  See V4.10.xx Release Notes for details.
   // V1.x, V2.x, and V3.x Revision History archived.
   // V4.00.00  2018-07-16:  Changed Inf_ items to HMI_, and added Cfg_Area for security.
   // Added Val_FirstOutTxt string (Local, read-only) for use in
   // IntlkTrip alarm message  (ref: KnowledgeBase answer ID 672568).
   // Deleted Cfg_PCmdClear; all Program Commands are now self-clearing.
   // All OCmds/MCmds and ORdys/MRdys are now Local Tags.
   // Added Sts_RdyReset for use by external objects.
   // V4.10.00  2019-03-08:  Changed type of Val_FirstOutTxt to STRING_Cond.
   // Corrected Scan Mode selection to execute Prescan logic. Added Cfg_HasMoreObj.\
   // V4.10.01  2019-10-16:  Modified conditions for clearing first-out status and text.
   // ============================================================
   // This Instruction monitors up to 16 Interlock conditions.  It provides these features:
   // *  The "OK" state of each Interlock Input is configurable.
   // By default, each Input is 1 to trip, 0 when OK to run.
   // *  Interlocks may be configured as Latched.  Latched Interlocks
   // require a Reset Command to clear.  The latching function can be inhibited
   // via a Latch Defeat input, for example, to avoid latching Interlocks for a stopped motor.
   // *  Interlocks may be configured as Bypassable.  Bypassable Interlocks are reported
   // separately; the destination object can use this information to bypass these
   // Interlocks in Maintenance Mode or upon command.
   // *  First-Out reporting indicates the first condition that
   // caused the running equipment to be tripped.
   // * For each Interlock condition, a Tag may be defined for navigation. Clicking
   // the Interlock description will call up the associated Tag's Faceplate.
   // ============================================================
   // SHOW LOCAL STRINGS
   // ============================================================
   // The STRINGs containing the text associated with each instance of this
   // instruction cannot be Input or Output Parameters, because STRINGs are not
   //  'atomic' types. (Inputs and Outputs must be SINT, INT, DINT, REAL, or BOOL.)
   // In order to make it easier to find and configure these STRINGs, this rung
   // was added.  THE JMP (and the LBL on the following rung)
   // MUST NOT BE REMOVED!!!
   // To view the STRINGs, go to the instruction instance (in LD or FBD), RIGHT-click
   // to bring up the context menu and select "Open Instruction Logic".
   // This rung will appear with the STRING values for the selected instance.
   // You may double-click the STRING values here to modify them as well.
   // #####  V4.00.00  2018-07-16:  Added string for Cfg_Area, Val_FirstOutTxt; renamed Inf_* to HMI_*.  #####
   0: JMP(SkipText)[LOWER(Cfg_Desc,Cfg_Label) LOWER(Cfg_Tag,Cfg_Area) CONCAT(HMI_Lib,HMI_Type,Val_FirstOutTxt) ,LOWER(Cfg_CondTxt[0],Cfg_CondTxt[1]) LOWER(Cfg_CondTxt[2],Cfg_CondTxt[3]) LOWER(Cfg_CondTxt[4],Cfg_CondTxt[5]) LOWER(Cfg_CondTxt[6],Cfg_CondTxt[7]) ,LOWER(Cfg_CondTxt[8],Cfg_CondTxt[9]) LOWER(Cfg_CondTxt[10],Cfg_CondTxt[11]) LOWER(Cfg_CondTxt[12],Cfg_CondTxt[13]) LOWER(Cfg_CondTxt[14],Cfg_CondTxt[15]) ,LOWER(Cfg_NavTag[0],Cfg_NavTag[1]) LOWER(Cfg_NavTag[2],Cfg_NavTag[3]) LOWER(Cfg_NavTag[4],Cfg_NavTag[5]) LOWER(Cfg_NavTag[6],Cfg_NavTag[7]) ,LOWER(Cfg_NavTag[8],Cfg_NavTag[9]) LOWER(Cfg_NavTag[10],Cfg_NavTag[11]) LOWER(Cfg_NavTag[12],Cfg_NavTag[13]) LOWER(Cfg_NavTag[14],Cfg_NavTag[15]) ];
   // ============================================================
   // INPUT GATHERING
   // ============================================================
   // This object uses word-wise logic.  The 16 interlock inputs are aliased
   // to the Wrk_Inp word, so no logic is needed to collect the individual
   // conditions.  We can immediately start processing the interlock logic.
   // ============================================================
   // HANDLE "OK STATE" INVERSIONS
   // ============================================================
   // This rung inverts the Input bits whose "OK State" is 1 (0 to Stop).
   // The resulting Wrk_Inp word is ZERO if all interlock inputs are "OK".
   1: LBL(SkipText)XOR(Wrk_Inp,Cfg_OKState,Wrk_InpInv);
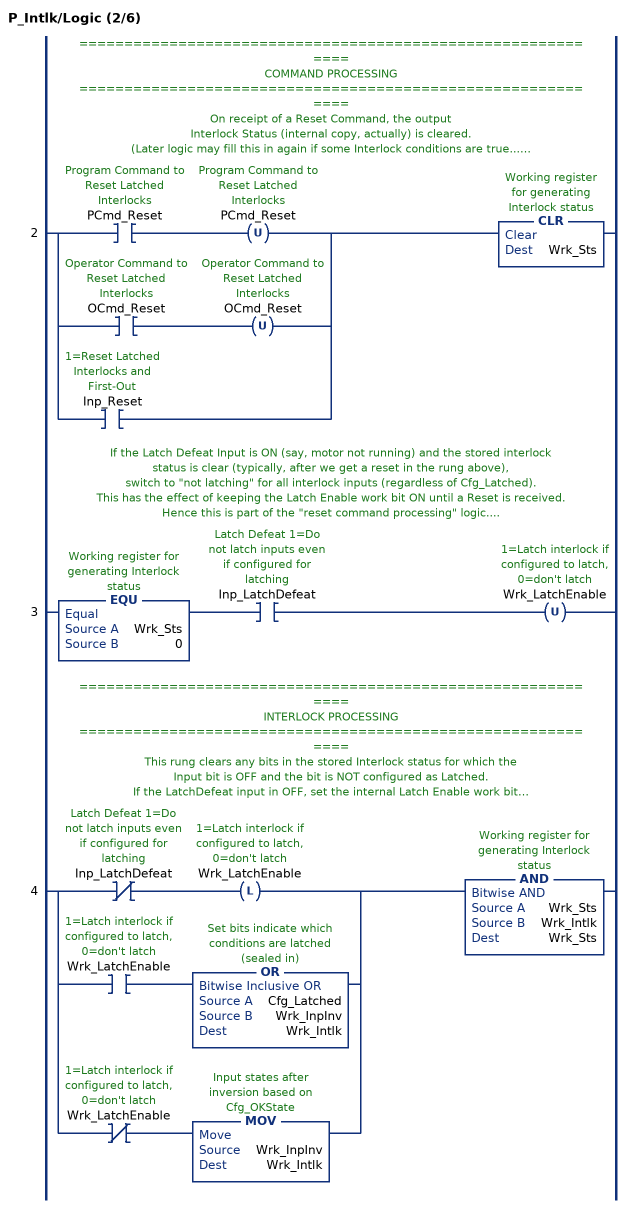
   // ============================================================
   // COMMAND PROCESSING
   // ============================================================
   // On receipt of a Reset Command, the output
   // Interlock Status (internal copy, actually) is cleared.
   // (Later logic may fill this in again if some Interlock conditions are true...)
   // NOTE:  This object is "Modeless" -- Operator and Program Commands
   // are accepted at any time.
   // #####  V4.00.00  2018-07-16:  Deleted Cfg_PCmdClear; all Program Commands are now self-clearing.  #####
   2: [XIC(PCmd_Reset) OTU(PCmd_Reset) ,XIC(OCmd_Reset) OTU(OCmd_Reset) ,XIC(Inp_Reset) ]CLR(Wrk_Sts);
   // If the Latch Defeat Input is ON (say, motor not running) and the stored interlock
   // status is clear (typically, after we get a reset in the rung above),
   // switch to "not latching" for all interlock inputs (regardless of Cfg_Latched).
   // This has the effect of keeping the Latch Enable work bit ON until a Reset is received.
   // Hence this is part of the "reset command processing" logic....
   3: EQU(Wrk_Sts,0)XIC(Inp_LatchDefeat)OTU(Wrk_LatchEnable);
   // ============================================================
   // INTERLOCK PROCESSING
   // ============================================================
   // This rung clears any bits in the stored Interlock status for which the
   // Input bit is OFF and the bit is NOT configured as Latched.
   // If the LatchDefeat input in OFF, set the internal Latch Enable work bit.
   // If this bit is ON, don't clear any latched bits with this rung (keep them latched).
   // If this bit is OFF, clear any bits that are NOT on in the input, whether
   // configured for latching or not!
   4: [XIO(Inp_LatchDefeat) OTL(Wrk_LatchEnable) ,XIC(Wrk_LatchEnable) OR(Cfg_Latched,Wrk_InpInv,Wrk_Intlk) ,XIO(Wrk_LatchEnable) MOV(Wrk_InpInv,Wrk_Intlk) ]AND(Wrk_Sts,Wrk_Intlk,Wrk_Sts);
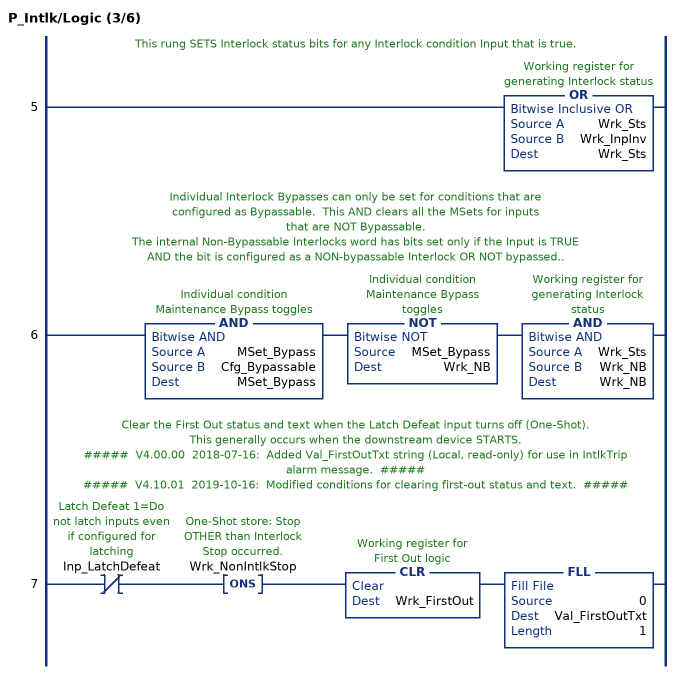
   // This rung SETS Interlock status bits for any Interlock condition Input that is true.
   5: OR(Wrk_Sts,Wrk_InpInv,Wrk_Sts);
   // Individual Interlock Bypasses can only be set for conditions that are
   // configured as Bypassable.  This AND clears all the MSets for inputs
   // that are NOT Bypassable.
   // The internal Non-Bypassable Interlocks word has bits set only if the Input is TRUE
   // AND the bit is configured as a NON-bypassable Interlock OR NOT bypassed..
   6: AND(MSet_Bypass,Cfg_Bypassable,MSet_Bypass)NOT(MSet_Bypass,Wrk_NB)AND(Wrk_Sts,Wrk_NB,Wrk_NB);
   // Clear the First Out status and text when the Latch Defeat input turns off (One-Shot).
   // This generally occurs when the downstream device STARTS.
   // #####  V4.00.00  2018-07-16:  Added Val_FirstOutTxt string (Local, read-only) for use in IntlkTrip alarm message.  #####
   // #####  V4.10.01  2019-10-16:  Modified conditions for clearing first-out status and text.  #####
   7: XIO(Inp_LatchDefeat)ONS(Wrk_NonIntlkStop)CLR(Wrk_FirstOut)FLL(0,Val_FirstOutTxt,1);
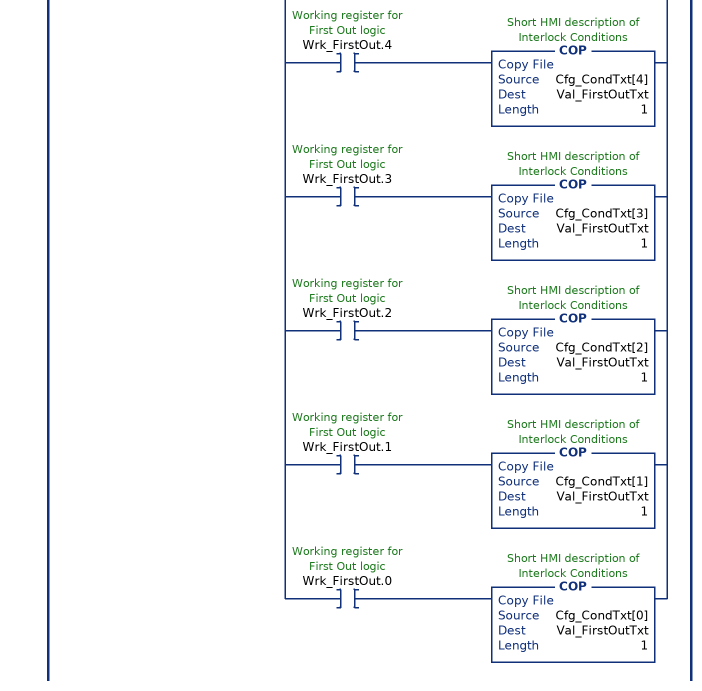
   // If an interlock condition occurs (which interlocks depends on the
   // bypass status!) and the Latch Defeat input is NOT set,
   // the equipment is running and will be shut down.
   // If this happens, record the First Out status.
   // #####  V4.00.00  2018-07-16:  Added Val_FirstOutTxt string (Local, read-only) for use in IntlkTrip alarm message.  #####
   // #####  V4.10.00  2019-03-08:  Changed type of Val_FirstOutTxt to STRING_Cond.  #####
   8: [XIO(Inp_BypActive) NEQ(Wrk_Sts,0) ,XIC(Inp_BypActive) NEQ(Wrk_NB,0) ]XIO(Inp_LatchDefeat)ONS(Wrk_SetFirstOut)[XIO(Inp_BypActive) CPT(Wrk_FirstOut,(Wrk_Sts)AND(NOT(Wrk_PrevSts))) ,XIC(Inp_BypActive) CPT(Wrk_FirstOut,(Wrk_NB)AND(NOT(Wrk_PrevSts))) ,NEQ(Wrk_FirstOut,0) [XIC(Wrk_FirstOut.15) COP(Cfg_CondTxt[15],Val_FirstOutTxt,1) ,XIC(Wrk_FirstOut.14) COP(Cfg_CondTxt[14],Val_FirstOutTxt,1) ,XIC(Wrk_FirstOut.13) COP(Cfg_CondTxt[13],Val_FirstOutTxt,1) ,XIC(Wrk_FirstOut.12) COP(Cfg_CondTxt[12],Val_FirstOutTxt,1) ,XIC(Wrk_FirstOut.11) COP(Cfg_CondTxt[11],Val_FirstOutTxt,1) ,XIC(Wrk_FirstOut.10) COP(Cfg_CondTxt[10],Val_FirstOutTxt,1) ,XIC(Wrk_FirstOut.9) COP(Cfg_CondTxt[9],Val_FirstOutTxt,1) ,XIC(Wrk_FirstOut.8) COP(Cfg_CondTxt[8],Val_FirstOutTxt,1) ,XIC(Wrk_FirstOut.7) COP(Cfg_CondTxt[7],Val_FirstOutTxt,1) ,XIC(Wrk_FirstOut.6) COP(Cfg_CondTxt[6],Val_FirstOutTxt,1) ,XIC(Wrk_FirstOut.5) COP(Cfg_CondTxt[5],Val_FirstOutTxt,1) ,XIC(Wrk_FirstOut.4) COP(Cfg_CondTxt[4],Val_FirstOutTxt,1) ,XIC(Wrk_FirstOut.3) COP(Cfg_CondTxt[3],Val_FirstOutTxt,1) ,XIC(Wrk_FirstOut.2) COP(Cfg_CondTxt[2],Val_FirstOutTxt,1) ,XIC(Wrk_FirstOut.1) COP(Cfg_CondTxt[1],Val_FirstOutTxt,1) ,XIC(Wrk_FirstOut.0) COP(Cfg_CondTxt[0],Val_FirstOutTxt,1) ] ];
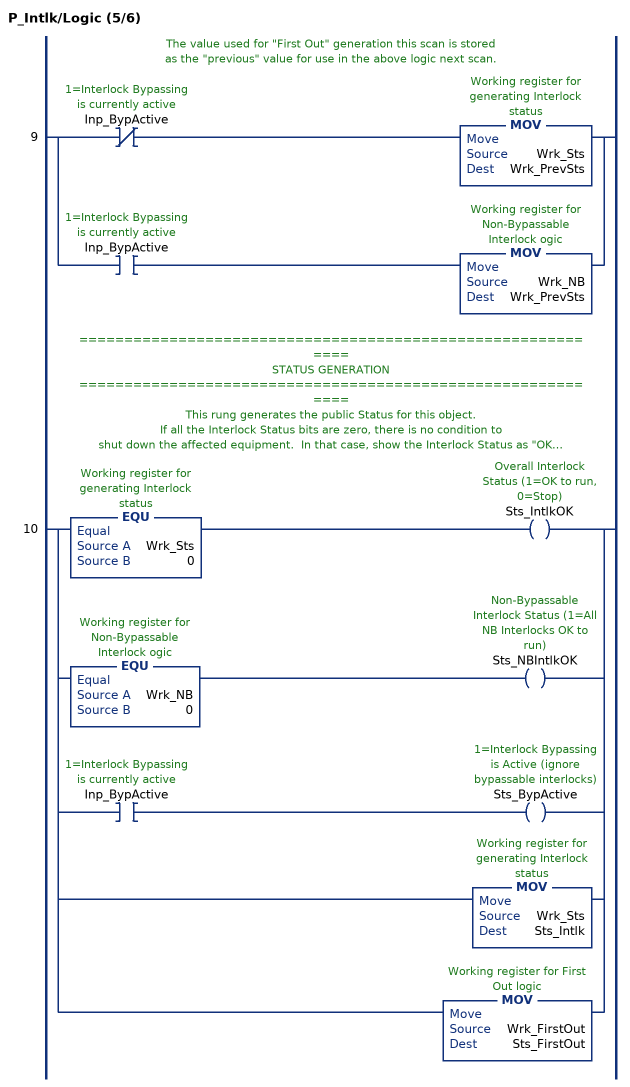
   // The value used for "First Out" generation this scan is stored
   // as the "previous" value for use in the above logic next scan.
   9: [XIO(Inp_BypActive) MOV(Wrk_Sts,Wrk_PrevSts) ,XIC(Inp_BypActive) MOV(Wrk_NB,Wrk_PrevSts) ];
   // ============================================================
   // STATUS GENERATION
   // ============================================================
   // This rung generates the public Status for this object.
   // If all the Interlock Status bits are zero, there is no condition to
   // shut down the affected equipment.  In that case, show the Interlock Status as "OK"
   // Similar logic applies for the Non-Bypassable Interlocks OK Status.
   // Also show the individual Interlock Status bits and the First Out Status bits.
   // NOTE:  Working registers are used to prevent outside writes to the Sts_xxx
   // parameters from affecting the state of this object!
   10: [[EQU(Wrk_Sts,0) OTE(Sts_IntlkOK) ,EQU(Wrk_NB,0) OTE(Sts_NBIntlkOK) ] ,XIC(Inp_BypActive) OTE(Sts_BypActive) ,MOV(Wrk_Sts,Sts_Intlk) ,MOV(Wrk_FirstOut,Sts_FirstOut) ];
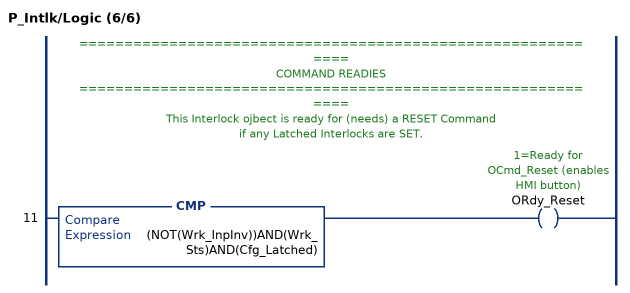
   // ============================================================
   // COMMAND READIES
   // ============================================================
   // This Interlock ojbect is ready for (needs) a RESET Command
   // if any Latched Interlocks are SET.
   11: CMP((NOT(Wrk_InpInv))AND(Wrk_Sts)AND(Cfg_Latched))OTE(ORdy_Reset);
END_ROUTINE
